// Brief: Slave Arm Endoscope Control
FUNCTION_BLOCK PUBLIC FB_SlaveCtrlEndoscope EXTENDS FB_SlaveArmCtrlBase
VAR_INPUT
END_VAR
VAR_OUTPUT
END_VAR
VAR
END_VAR

END_FUNCTION_BLOCK

(* stored: Version 1.1.0.1, ProductVersion 3.1.4024.12
   POU FB_SlaveCtrlEndoscope: Id {6b490525-446d-48f2-ab19-237faca074bd}, SpecialFunc None *)
